LIN {X 0,Y 100.402,Z 358.237,A -85,B 0,C 180,E1 -29156.99,E2 -29156.99} C_VEL
LIN {X 0,Y 100.384,Z 357.85,A -85,B 0,C 180,E1 -29157.993,E2 -29157.993} C_VEL
LIN {X 0,Y 100.386,Z 357.819,A -85,B 0,C 180,E1 -29161.253,E2 -29161.253} C_VEL
LIN {X 0,Y 101.796,Z 362.471,A -85,B 0,C 180,E1 -29171.07,E2 -29171.07} C_VEL
LIN {X 0,Y 103.401,Z 366.135,A -85,B 0,C 180,E1 -29175.775,E2 -29175.775} C_VEL
LIN {X 0,Y 105.074,Z 370.255,A -85,B 0,C 180,E1 -29179.684,E2 -29179.684} C_VEL
LIN {X 0,Y 105.684,Z 372.499,A -85,B 0,C 180,E1 -29181.129,E2 -29181.129} C_VEL
LIN {X 0,Y 106.021,Z 374.366,A -85,B 0,C 180,E1 -29182.034,E2 -29182.034} C_VEL
LIN {X 0,Y 103.387,Z 386.289,A -85,B 0,C 180,E1 -29182.916,E2 -29182.916} C_VEL
LIN {X 0,Y 99.941,Z 396.229,A -85,B 0,C 180,E1 -29183.916,E2 -29183.916} C_VEL
LIN {X 0,Y 96.046,Z 404.883,A -85,B 0,C 180,E1 -29185.113,E2 -29185.113} C_VEL
LIN {X 0,Y 91.456,Z 413.164,A -85,B 0,C 180,E1 -29186.711,E2 -29186.711} C_VEL
LIN {X 0,Y 86.224,Z 421.013,A -85,B 0,C 180,E1 -29188.816,E2 -29188.816} C_VEL
LIN {X 0,Y 80.026,Z 428.854,A -85,B 0,C 180,E1 -29191.798,E2 -29191.798} C_VEL
LIN {X 0,Y 72.277,Z 437.075,A -85,B 0,C 180,E1 -29196.664,E2 -29196.664} C_VEL
LIN {X 0,Y 65.93,Z 442.65,A -85,B 0,C 180,E1 -29201.744,E2 -29201.744} C_VEL
LIN {X 0,Y 59.276,Z 447.852,A -85,B 0,C 180,E1 -29209.305,E2 -29209.305} C_VEL
LIN {X 0,Y 53.929,Z 451.685,A -85,B 0,C 180,E1 -29218.587,E2 -29218.587} C_VEL
LIN {X 0,Y 51.351,Z 453.456,A -85,B 0,C 180,E1 -29225.763,E2 -29225.763} C_VEL
LIN {X 0,Y 49.572,Z 454.73,A -85,B 0,C 180,E1 -29233.533,E2 -29233.533} C_VEL
LIN {X 0,Y 48.724,Z 455.53,A -85,B 0,C 180,E1 -29241.711,E2 -29241.711} C_VEL
LIN {X 0,Y 48.789,Z 455.849,A -85,B 0,C 180,E1 -29250.004,E2 -29250.004} C_VEL
LIN {X 0,Y 48.725,Z 455.516,A -85,B 0,C 180,E1 -29258.297,E2 -29258.297} C_VEL
LIN {X 0,Y 49.574,Z 454.686,A -85,B 0,C 180,E1 -29266.476,E2 -29266.476} C_VEL
LIN {X 0,Y 51.352,Z 453.382,A -85,B 0,C 180,E1 -29274.245,E2 -29274.245} C_VEL
LIN {X 0,Y 55.511,Z 450.407,A -85,B 0,C 180,E1 -29284.736,E2 -29284.736} C_VEL
LIN {X 0,Y 59.279,Z 447.714,A -85,B 0,C 180,E1 -29290.702,E2 -29290.702} C_VEL
LIN {X 0,Y 65.928,Z 442.473,A -85,B 0,C 180,E1 -29298.267,E2 -29298.267} C_VEL
LIN {X 0,Y 73.597,Z 435.578,A -85,B 0,C 180,E1 -29304.266,E2 -29304.266} C_VEL
LIN {X 0,Y 80.378,Z 428.151,A -85,B 0,C 180,E1 -29308.358,E2 -29308.358} C_VEL
LIN {X 0,Y 85.511,Z 421.674,A -85,B 0,C 180,E1 -29310.843,E2 -29310.843} C_VEL
LIN {X 0,Y 90.682,Z 413.947,A -85,B 0,C 180,E1 -29313.038,E2 -29313.038} C_VEL
LIN {X 0,Y 95.26,Z 405.834,A -85,B 0,C 180,E1 -29314.663,E2 -29314.663} C_VEL
LIN {X 0,Y 99.139,Z 397.416,A -85,B 0,C 180,E1 -29315.887,E2 -29315.887} C_VEL
LIN {X 0,Y 102.671,Z 387.658,A -85,B 0,C 180,E1 -29316.868,E2 -29316.868} C_VEL
LIN {X 0,Y 105.515,Z 376.095,A -85,B 0,C 180,E1 -29317.75,E2 -29317.75} C_VEL
LIN {X 0,Y 105.767,Z 374.04,A -85,B 0,C 180,E1 -29317.928,E2 -29317.928} C_VEL
LIN {X 0,Y 105.084,Z 370.805,A -85,B 0,C 180,E1 -29319.661,E2 -29319.661} C_VEL
LIN {X 0,Y 103.427,Z 366.583,A -85,B 0,C 180,E1 -29323.437,E2 -29323.437} C_VEL
LIN {X 0,Y 102.311,Z 364.174,A -85,B 0,C 180,E1 -29326.284,E2 -29326.284} C_VEL
LIN {X 0,Y 101.255,Z 361.634,A -85,B 0,C 180,E1 -29329.818,E2 -29329.818} C_VEL
LIN {X 0,Y 100.146,Z 358.287,A -85,B 0,C 180,E1 -29336.732,E2 -29336.732} C_VEL
LIN {X 0,Y 100.091,Z 357.785,A -85,B 0,C 180,E1 -29337.988,E2 -29337.988} C_VEL
LIN {X 0,Y 100.101,Z 357.82,A -85,B 0,C 180,E1 -29343.019,E2 -29343.019} C_VEL
LIN {X 0,Y 101.129,Z 361.456,A -85,B 0,C 180,E1 -29350.546,E2 -29350.546} C_VEL
LIN {X 0,Y 101.708,Z 362.817,A -85,B 0,C 180,E1 -29352.682,E2 -29352.682} C_VEL
LIN {X 0,Y 103.187,Z 366.252,A -85,B 0,C 180,E1 -29357.049,E2 -29357.049} C_VEL
LIN {X 0,Y 104.694,Z 370.111,A -85,B 0,C 180,E1 -29360.703,E2 -29360.703} C_VEL
LIN {X 0,Y 105.664,Z 373.274,A -85,B 0,C 180,E1 -29363.045,E2 -29363.045} C_VEL
LIN {X 0,Y 103.161,Z 383.593,A -85,B 0,C 180,E1 -29364.046,E2 -29364.046} C_VEL
LIN {X 0,Y 100.108,Z 392.746,A -85,B 0,C 180,E1 -29365.323,E2 -29365.323} C_VEL
LIN {X 0,Y 96.36,Z 401.138,A -85,B 0,C 180,E1 -29366.686,E2 -29366.686} C_VEL
LIN {X 0,Y 92.666,Z 407.987,A -85,B 0,C 180,E1 -29368.152,E2 -29368.152} C_VEL
LIN {X 0,Y 87.652,Z 415.86,A -85,B 0,C 180,E1 -29370.461,E2 -29370.461} C_VEL
LIN {X 0,Y 83.407,Z 421.515,A -85,B 0,C 180,E1 -29372.578,E2 -29372.578} C_VEL
LIN {X 0,Y 77.628,Z 428.233,A -85,B 0,C 180,E1 -29376.073,E2 -29376.073} C_VEL
LIN {X 0,Y 73.727,Z 431.905,A -85,B 0,C 180,E1 -29378.076,E2 -29378.076} C_VEL
LIN {X 0,Y 66.062,Z 437.234,A -85,B 0,C 180,E1 -29380.871,E2 -29380.871} C_VEL
LIN {X 0,Y 58.269,Z 441.79,A -85,B 0,C 180,E1 -29384.678,E2 -29384.678} C_VEL
LIN {X 0,Y 54.358,Z 444.075,A -85,B 0,C 180,E1 -29388.459,E2 -29388.459} C_VEL
LIN {X 0,Y 49.897,Z 446.751,A -85,B 0,C 180,E1 -29395.704,E2 -29395.704} C_VEL
LIN {X 0,Y 46.656,Z 448.491,A -85,B 0,C 180,E1 -29403.129,E2 -29403.129} C_VEL
LIN {X 0,Y 44.155,Z 449.745,A -85,B 0,C 180,E1 -29411.433,E2 -29411.433} C_VEL
LIN {X 0,Y 42.609,Z 450.532,A -85,B 0,C 180,E1 -29420.501,E2 -29420.501} C_VEL
LIN {X 0,Y 42.085,Z 450.831,A -85,B 0,C 180,E1 -29429.995,E2 -29429.995} C_VEL
LIN {X 0,Y 42.608,Z 450.55,A -85,B 0,C 180,E1 -29439.489,E2 -29439.489} C_VEL
LIN {X 0,Y 44.15,Z 449.799,A -85,B 0,C 180,E1 -29448.559,E2 -29448.559} C_VEL
LIN {X 0,Y 46.62,Z 448.583,A -85,B 0,C 180,E1 -29456.883,E2 -29456.883} C_VEL
LIN {X 0,Y 51.76,Z 445.741,A -85,B 0,C 180,E1 -29467.657,E2 -29467.657} C_VEL
LIN {X 0,Y 55.967,Z 443.15,A -85,B 0,C 180,E1 -29473.677,E2 -29473.677} C_VEL
LIN {X 0,Y 63.208,Z 438.053,A -85,B 0,C 180,E1 -29481.102,E2 -29481.102} C_VEL
LIN {X 0,Y 69.847,Z 432.563,A -85,B 0,C 180,E1 -29486.105,E2 -29486.105} C_VEL
LIN {X 0,Y 76.92,Z 425.648,A -85,B 0,C 180,E1 -29490.221,E2 -29490.221} C_VEL
LIN {X 0,Y 83.481,Z 417.714,A -85,B 0,C 180,E1 -29493.436,E2 -29493.436} C_VEL
LIN {X 0,Y 88.75,Z 410.141,A -85,B 0,C 180,E1 -29495.591,E2 -29495.591} C_VEL
LIN {X 0,Y 92.616,Z 403.681,A -85,B 0,C 180,E1 -29496.932,E2 -29496.932} C_VEL
LIN {X 0,Y 96.47,Z 395.828,A -85,B 0,C 180,E1 -29498.251,E2 -29498.251} C_VEL
LIN {X 0,Y 99.737,Z 387.4,A -85,B 0,C 180,E1 -29499.37,E2 -29499.37} C_VEL
LIN {X 0,Y 102.526,Z 377.614,A -85,B 0,C 180,E1 -29500.363,E2 -29500.363} C_VEL
LIN {X 0,Y 102.555,Z 376.884,A -85,B 0,C 180,E1 -29500.653,E2 -29500.653} C_VEL
LIN {X 0,Y 101.635,Z 373.042,A -85,B 0,C 180,E1 -29504.329,E2 -29504.329} C_VEL
LIN {X 0,Y 100.893,Z 370.848,A -85,B 0,C 180,E1 -29507.018,E2 -29507.018} C_VEL
LIN {X 0,Y 100.114,Z 368.403,A -85,B 0,C 180,E1 -29510.657,E2 -29510.657} C_VEL
LIN {X 0,Y 99.502,Z 364.863,A -85,B 0,C 180,E1 -29518.482,E2 -29518.482} C_VEL
LIN {X 0,Y 99.503,Z 365.013,A -85,B 0,C 180,E1 -29521.264,E2 -29521.264} C_VEL
LIN {X 0,Y 100.461,Z 369.199,A -85,B 0,C 180,E1 -29529.945,E2 -29529.945} C_VEL
LIN {X 0,Y 101.631,Z 372.591,A -85,B 0,C 180,E1 -29534.377,E2 -29534.377} C_VEL
LIN {X 0,Y 102.921,Z 376.479,A -85,B 0,C 180,E1 -29538.153,E2 -29538.153} C_VEL
LIN {X 0,Y 103.002,Z 377.05,A -85,B 0,C 180,E1 -29538.524,E2 -29538.524} C_VEL
LIN {X 0,Y 100.454,Z 387.016,A -85,B 0,C 180,E1 -29539.275,E2 -29539.275} C_VEL
LIN {X 0,Y 97.284,Z 395.844,A -85,B 0,C 180,E1 -29540.099,E2 -29540.099} C_VEL
LIN {X 0,Y 93.252,Z 404.495,A -85,B 0,C 180,E1 -29541.155,E2 -29541.155} C_VEL
LIN {X 0,Y 88.492,Z 412.776,A -85,B 0,C 180,E1 -29542.601,E2 -29542.601} C_VEL
LIN {X 0,Y 83.033,Z 420.624,A -85,B 0,C 180,E1 -29544.516,E2 -29544.516} C_VEL
LIN {X 0,Y 77.068,Z 427.848,A -85,B 0,C 180,E1 -29547.032,E2 -29547.032} C_VEL
LIN {X 0,Y 69.679,Z 435.442,A -85,B 0,C 180,E1 -29550.988,E2 -29550.988} C_VEL
LIN {X 0,Y 62.724,Z 441.292,A -85,B 0,C 180,E1 -29555.681,E2 -29555.681} C_VEL
LIN {X 0,Y 56.429,Z 445.925,A -85,B 0,C 180,E1 -29561.65,E2 -29561.65} C_VEL
LIN {X 0,Y 51.851,Z 448.938,A -85,B 0,C 180,E1 -29567.341,E2 -29567.341} C_VEL
LIN {X 0,Y 47.976,Z 451.291,A -85,B 0,C 180,E1 -29574.135,E2 -29574.135} C_VEL
LIN {X 0,Y 44.947,Z 453.063,A -85,B 0,C 180,E1 -29582.031,E2 -29582.031} C_VEL
LIN {X 0,Y 42.797,Z 454.337,A -85,B 0,C 180,E1 -29590.832,E2 -29590.832} C_VEL
LIN {X 0,Y 41.689,Z 455.137,A -85,B 0,C 180,E1 -29600.3,E2 -29600.3} C_VEL
LIN {X 0,Y 41.692,Z 455.457,A -85,B 0,C 180,E1 -29610.005,E2 -29610.005} C_VEL
LIN {X 0,Y 41.69,Z 455.122,A -85,B 0,C 180,E1 -29619.71,E2 -29619.71} C_VEL
LIN {X 0,Y 42.799,Z 454.293,A -85,B 0,C 180,E1 -29629.178,E2 -29629.178} C_VEL
LIN {X 0,Y 44.949,Z 452.988,A -85,B 0,C 180,E1 -29637.979,E2 -29637.979} C_VEL
LIN {X 0,Y 49.822,Z 450.012,A -85,B 0,C 180,E1 -29649.408,E2 -29649.408} C_VEL
LIN {X 0,Y 54.09,Z 447.321,A -85,B 0,C 180,E1 -29655.618,E2 -29655.618} C_VEL
LIN {X 0,Y 61.408,Z 442.077,A -85,B 0,C 180,E1 -29663.244,E2 -29663.244} C_VEL
LIN {X 0,Y 69.684,Z 435.183,A -85,B 0,C 180,E1 -29669.017,E2 -29669.017} C_VEL
LIN {X 0,Y 75.984,Z 428.786,A -85,B 0,C 180,E1 -29672.454,E2 -29672.454} C_VEL
LIN {X 0,Y 82.27,Z 421.277,A -85,B 0,C 180,E1 -29675.189,E2 -29675.189} C_VEL
LIN {X 0,Y 87.699,Z 413.553,A -85,B 0,C 180,E1 -29677.165,E2 -29677.165} C_VEL
LIN {X 0,Y 92.44,Z 405.437,A -85,B 0,C 180,E1 -29678.65,E2 -29678.65} C_VEL
LIN {X 0,Y 96.462,Z 397.019,A -85,B 0,C 180,E1 -29679.731,E2 -29679.731} C_VEL
LIN {X 0,Y 99.499,Z 389.051,A -85,B 0,C 180,E1 -29680.457,E2 -29680.457} C_VEL
LIN {X 0,Y 102.181,Z 379.433,A -85,B 0,C 180,E1 -29681.182,E2 -29681.182} C_VEL
LIN {X 0,Y 102.772,Z 376.736,A -85,B 0,C 180,E1 -29681.433,E2 -29681.433} C_VEL
LIN {X 0,Y 101.62,Z 373.025,A -85,B 0,C 180,E1 -29684.789,E2 -29684.789} C_VEL
LIN {X 0,Y 100.366,Z 369.551,A -85,B 0,C 180,E1 -29689.153,E2 -29689.153} C_VEL
LIN {X 0,Y 99.916,Z 368.232,A -85,B 0,C 180,E1 -29691.277,E2 -29691.277} C_VEL
LIN {X 0,Y 99.189,Z 364.754,A -85,B 0,C 180,E1 -29698.732,E2 -29698.732} C_VEL
LIN {X 0,Y 99.202,Z 364.859,A -85,B 0,C 180,E1 -29702.538,E2 -29702.538} C_VEL
LIN {X 0,Y 99.869,Z 368.268,A -85,B 0,C 180,E1 -29709.696,E2 -29709.696} C_VEL
LIN {X 0,Y 101.258,Z 372.35,A -85,B 0,C 180,E1 -29715.354,E2 -29715.354} C_VEL
LIN {X 0,Y 102.29,Z 376.488,A -85,B 0,C 180,E1 -29719.379,E2 -29719.379} C_VEL
LIN {X 0,Y 102.337,Z 377.035,A -85,B 0,C 180,E1 -29719.71,E2 -29719.71} C_VEL
LIN {X 0,Y 100.312,Z 384.55,A -85,B 0,C 180,E1 -29720.425,E2 -29720.425} C_VEL
LIN {X 0,Y 97.025,Z 393.794,A -85,B 0,C 180,E1 -29721.647,E2 -29721.647} C_VEL
LIN {X 0,Y 93.39,Z 401.547,A -85,B 0,C 180,E1 -29722.807,E2 -29722.807} C_VEL
LIN {X 0,Y 89.544,Z 408.381,A -85,B 0,C 180,E1 -29724.155,E2 -29724.155} C_VEL
LIN {X 0,Y 84.281,Z 416.255,A -85,B 0,C 180,E1 -29726.304,E2 -29726.304} C_VEL
LIN {X 0,Y 79.813,Z 421.909,A -85,B 0,C 180,E1 -29728.286,E2 -29728.286} C_VEL
LIN {X 0,Y 74.088,Z 428.217,A -85,B 0,C 180,E1 -29731.374,E2 -29731.374} C_VEL
LIN {X 0,Y 68.527,Z 433.462,A -85,B 0,C 180,E1 -29734.864,E2 -29734.864} C_VEL
LIN {X 0,Y 63.252,Z 437.837,A -85,B 0,C 180,E1 -29738.938,E2 -29738.938} C_VEL
LIN {X 0,Y 55.986,Z 442.983,A -85,B 0,C 180,E1 -29746.332,E2 -29746.332} C_VEL
LIN {X 0,Y 54.358,Z 444.075,A -85,B 0,C 180,E1 -29748.459,E2 -29748.459} C_VEL
LIN {X 0,Y 50.637,Z 446.185,A -85,B 0,C 180,E1 -29752.92,E2 -29752.92} C_VEL
LIN {X 0,Y 46.435,Z 447.925,A -85,B 0,C 180,E1 -29757.46,E2 -29757.46} C_VEL
LIN {X 0,Y 38.447,Z 450.266,A -85,B 0,C 180,E1 -29769.13,E2 -29769.13} C_VEL
LIN {X 0,Y 35.883,Z 450.882,A -85,B 0,C 180,E1 -29777.367,E2 -29777.367} C_VEL
LIN {X 0,Y 35.442,Z 450.973,A -85,B 0,C 180,E1 -29780.47,E2 -29780.47} C_VEL
LIN {X 0,Y 34.998,Z 451.223,A -85,B 0,C 180,E1 -29789.994,E2 -29789.994} C_VEL
LIN {X 0,Y 35.643,Z 450.94,A -85,B 0,C 180,E1 -29801.366,E2 -29801.366} C_VEL
LIN {X 0,Y 37.52,Z 450.189,A -85,B 0,C 180,E1 -29811.995,E2 -29811.995} C_VEL
LIN {X 0,Y 40.426,Z 448.974,A -85,B 0,C 180,E1 -29821.429,E2 -29821.429} C_VEL
LIN {X 0,Y 46.354,Z 446.131,A -85,B 0,C 180,E1 -29833.015,E2 -29833.015} C_VEL
LIN {X 0,Y 51.071,Z 443.54,A -85,B 0,C 180,E1 -29839.182,E2 -29839.182} C_VEL
LIN {X 0,Y 59.02,Z 438.442,A -85,B 0,C 180,E1 -29846.458,E2 -29846.458} C_VEL
LIN {X 0,Y 66.162,Z 432.952,A -85,B 0,C 180,E1 -29851.198,E2 -29851.198} C_VEL
LIN {X 0,Y 73.66,Z 426.037,A -85,B 0,C 180,E1 -29855.005,E2 -29855.005} C_VEL
LIN {X 0,Y 80.569,Z 418.101,A -85,B 0,C 180,E1 -29857.936,E2 -29857.936} C_VEL
LIN {X 0,Y 86.069,Z 410.528,A -85,B 0,C 180,E1 -29859.882,E2 -29859.882} C_VEL
LIN {X 0,Y 90.049,Z 404.122,A -85,B 0,C 180,E1 -29861.069,E2 -29861.069} C_VEL
LIN {X 0,Y 94.343,Z 395.59,A -85,B 0,C 180,E1 -29862.338,E2 -29862.338} C_VEL
LIN {X 0,Y 97.85,Z 386.64,A -85,B 0,C 180,E1 -29863.37,E2 -29863.37} C_VEL
LIN {X 0,Y 99.213,Z 382.499,A -85,B 0,C 180,E1 -29863.788,E2 -29863.788} C_VEL
LIN {X 0,Y 99.604,Z 380.632,A -85,B 0,C 180,E1 -29864.263,E2 -29864.263} C_VEL
LIN {X 0,Y 98.889,Z 377.185,A -85,B 0,C 180,E1 -29868.446,E2 -29868.446} C_VEL
LIN {X 0,Y 98.533,Z 375.072,A -85,B 0,C 180,E1 -29871.798,E2 -29871.798} C_VEL
LIN {X 0,Y 98.345,Z 371.862,A -85,B 0,C 180,E1 -29878.976,E2 -29878.976} C_VEL
LIN {X 0,Y 98.338,Z 371.997,A -85,B 0,C 180,E1 -29880.639,E2 -29880.639} C_VEL
LIN {X 0,Y 98.892,Z 375.878,A -85,B 0,C 180,E1 -29888.814,E2 -29888.814} C_VEL
LIN {X 0,Y 99.577,Z 378.924,A -85,B 0,C 180,E1 -29893.001,E2 -29893.001} C_VEL
LIN {X 0,Y 99.979,Z 380.711,A -85,B 0,C 180,E1 -29894.939,E2 -29894.939} C_VEL
LIN {X 0,Y 97.288,Z 389.687,A -85,B 0,C 180,E1 -29895.575,E2 -29895.575} C_VEL
LIN {X 0,Y 93.418,Z 399.209,A -85,B 0,C 180,E1 -29896.43,E2 -29896.43} C_VEL
LIN {X 0,Y 87.642,Z 409.922,A -85,B 0,C 180,E1 -29897.786,E2 -29897.786} C_VEL
LIN {X 0,Y 81.96,Z 418.188,A -85,B 0,C 180,E1 -29899.406,E2 -29899.406} C_VEL
LIN {X 0,Y 75.571,Z 425.873,A -85,B 0,C 180,E1 -29901.575,E2 -29901.575} C_VEL
LIN {X 0,Y 69.317,Z 432.203,A -85,B 0,C 180,E1 -29904.154,E2 -29904.154} C_VEL
LIN {X 0,Y 63.294,Z 437.474,A -85,B 0,C 180,E1 -29907.347,E2 -29907.347} C_VEL
LIN {X 0,Y 57.427,Z 441.865,A -85,B 0,C 180,E1 -29911.063,E2 -29911.063} C_VEL
LIN {X 0,Y 49.379,Z 447.07,A -85,B 0,C 180,E1 -29918.489,E2 -29918.489} C_VEL
LIN {X 0,Y 42.397,Z 450.898,A -85,B 0,C 180,E1 -29928.473,E2 -29928.473} C_VEL
LIN {X 0,Y 38.782,Z 452.669,A -85,B 0,C 180,E1 -29937.074,E2 -29937.074} C_VEL
LIN {X 0,Y 36.161,Z 453.945,A -85,B 0,C 180,E1 -29947.133,E2 -29947.133} C_VEL
LIN {X 0,Y 34.707,Z 454.745,A -85,B 0,C 180,E1 -29958.323,E2 -29958.323} C_VEL
LIN {X 0,Y 34.585,Z 455.065,A -85,B 0,C 180,E1 -29970.006,E2 -29970.006} C_VEL
LIN {X 0,Y 34.709,Z 454.73,A -85,B 0,C 180,E1 -29981.688,E2 -29981.688} C_VEL
LIN {X 0,Y 36.163,Z 453.9,A -85,B 0,C 180,E1 -29992.878,E2 -29992.878} C_VEL
LIN {X 0,Y 38.784,Z 452.593,A -85,B 0,C 180,E1 -30002.937,E2 -30002.937} C_VEL
LIN {X 0,Y 44.555,Z 449.619,A -85,B 0,C 180,E1 -30015.227,E2 -30015.227} C_VEL
LIN {X 0,Y 49.383,Z 446.927,A -85,B 0,C 180,E1 -30021.519,E2 -30021.519} C_VEL
LIN {X 0,Y 57.428,Z 441.682,A -85,B 0,C 180,E1 -30028.95,E2 -30028.95} C_VEL
LIN {X 0,Y 66.3,Z 434.788,A -85,B 0,C 180,E1 -30034.299,E2 -30034.299} C_VEL
LIN {X 0,Y 73.739,Z 427.556,A -85,B 0,C 180,E1 -30037.71,E2 -30037.71} C_VEL
LIN {X 0,Y 79.547,Z 420.881,A -85,B 0,C 180,E1 -30039.845,E2 -30039.845} C_VEL
LIN {X 0,Y 85.195,Z 413.157,A -85,B 0,C 180,E1 -30041.569,E2 -30041.569} C_VEL
LIN {X 0,Y 90.102,Z 405.041,A -85,B 0,C 180,E1 -30042.851,E2 -30042.851} C_VEL
LIN {X 0,Y 94.245,Z 396.622,A -85,B 0,C 180,E1 -30043.77,E2 -30043.77} C_VEL
LIN {X 0,Y 97.61,Z 387.893,A -85,B 0,C 180,E1 -30044.461,E2 -30044.461} C_VEL
LIN {X 0,Y 99.726,Z 380.373,A -85,B 0,C 180,E1 -30045.074,E2 -30045.074} C_VEL
LIN {X 0,Y 98.946,Z 377.09,A -85,B 0,C 180,E1 -30048.996,E2 -30048.996} C_VEL
LIN {X 0,Y 98.423,Z 374.847,A -85,B 0,C 180,E1 -30052.564,E2 -30052.564} C_VEL
LIN {X 0,Y 98.038,Z 371.726,A -85,B 0,C 180,E1 -30059.359,E2 -30059.359} C_VEL
LIN {X 0,Y 98.008,Z 371.971,A -85,B 0,C 180,E1 -30062.055,E2 -30062.055} C_VEL
LIN {X 0,Y 98.409,Z 375.692,A -85,B 0,C 180,E1 -30069.841,E2 -30069.841} C_VEL
LIN {X 0,Y 99.023,Z 378.8,A -85,B 0,C 180,E1 -30074.122,E2 -30074.122} C_VEL
LIN {X 0,Y 99.351,Z 380.461,A -85,B 0,C 180,E1 -30075.91,E2 -30075.91} C_VEL
LIN {X 0,Y 98.07,Z 384.948,A -85,B 0,C 180,E1 -30076.555,E2 -30076.555} C_VEL
LIN {X 0,Y 95.174,Z 392.928,A -85,B 0,C 180,E1 -30077.485,E2 -30077.485} C_VEL
LIN {X 0,Y 91.504,Z 400.808,A -85,B 0,C 180,E1 -30078.543,E2 -30078.543} C_VEL
LIN {X 0,Y 86.888,Z 408.776,A -85,B 0,C 180,E1 -30079.892,E2 -30079.892} C_VEL
LIN {X 0,Y 81.394,Z 416.649,A -85,B 0,C 180,E1 -30081.835,E2 -30081.835} C_VEL
LIN {X 0,Y 76.711,Z 422.303,A -85,B 0,C 180,E1 -30083.622,E2 -30083.622} C_VEL
LIN {X 0,Y 70.657,Z 428.611,A -85,B 0,C 180,E1 -30086.46,E2 -30086.46} C_VEL
LIN {X 0,Y 64.743,Z 433.855,A -85,B 0,C 180,E1 -30089.719,E2 -30089.719} C_VEL
LIN {X 0,Y 59.057,Z 438.23,A -85,B 0,C 180,E1 -30093.584,E2 -30093.584} C_VEL
LIN {X 0,Y 51.089,Z 443.376,A -85,B 0,C 180,E1 -30100.829,E2 -30100.829} C_VEL
LIN {X 0,Y 46.37,Z 446.006,A -85,B 0,C 180,E1 -30106.991,E2 -30106.991} C_VEL
LIN {X 0,Y 40.472,Z 448.882,A -85,B 0,C 180,E1 -30118.598,E2 -30118.598} C_VEL
LIN {X 0,Y 37.525,Z 450.136,A -85,B 0,C 180,E1 -30127.996,E2 -30127.996} C_VEL
LIN {X 0,Y 35.442,Z 450.973,A -85,B 0,C 180,E1 -30140.47,E2 -30140.47} C_VEL
LIN {X 0,Y 34.306,Z 451.261,A -85,B 0,C 180,E1 -30150.01,E2 -30150.01} C_VEL
LIN {X 0,Y 32.738,Z 450.99,A -85,B 0,C 180,E1 -30166.819,E2 -30166.819} C_VEL
LIN {X 0,Y 33.895,Z 449.832,A -85,B 0,C 180,E1 -30183.784,E2 -30183.784} C_VEL
LIN {X 0,Y 36.683,Z 448.514,A -85,B 0,C 180,E1 -30192.088,E2 -30192.088} C_VEL
LIN {X 0,Y 44.037,Z 445.376,A -85,B 0,C 180,E1 -30202.927,E2 -30202.927} C_VEL
LIN {X 0,Y 52.467,Z 440.726,A -85,B 0,C 180,E1 -30210.529,E2 -30210.529} C_VEL
LIN {X 0,Y 59.967,Z 435.669,A -85,B 0,C 180,E1 -30215.26,E2 -30215.26} C_VEL
LIN {X 0,Y 66.199,Z 430.719,A -85,B 0,C 180,E1 -30218.261,E2 -30218.261} C_VEL
LIN {X 0,Y 72.547,Z 424.746,A -85,B 0,C 180,E1 -30220.817,E2 -30220.817} C_VEL
LIN {X 0,Y 78.999,Z 417.473,A -85,B 0,C 180,E1 -30223,E2 -30223} C_VEL
LIN {X 0,Y 84.726,Z 409.689,A -85,B 0,C 180,E1 -30224.631,E2 -30224.631} C_VEL
LIN {X 0,Y 88.649,Z 403.371,A -85,B 0,C 180,E1 -30225.551,E2 -30225.551} C_VEL
LIN {X 0,Y 92.898,Z 394.941,A -85,B 0,C 180,E1 -30226.638,E2 -30226.638} C_VEL
LIN {X 0,Y 96.367,Z 386.136,A -85,B 0,C 180,E1 -30227.495,E2 -30227.495} C_VEL
LIN {X 0,Y 96.702,Z 384.376,A -85,B 0,C 180,E1 -30228.471,E2 -30228.471} C_VEL
LIN {X 0,Y 96.608,Z 382.315,A -85,B 0,C 180,E1 -30231.634,E2 -30231.634} C_VEL
LIN {X 0,Y 96.667,Z 379.04,A -85,B 0,C 180,E1 -30238.958,E2 -30238.958} C_VEL
LIN {X 0,Y 96.696,Z 378.99,A -85,B 0,C 180,E1 -30240.26,E2 -30240.26} C_VEL
LIN {X 0,Y 96.851,Z 382.493,A -85,B 0,C 180,E1 -30247.819,E2 -30247.819} C_VEL
LIN {X 0,Y 97.126,Z 384.2,A -85,B 0,C 180,E1 -30250.424,E2 -30250.424} C_VEL
LIN {X 0,Y 96.746,Z 386.119,A -85,B 0,C 180,E1 -30251.302,E2 -30251.302} C_VEL
LIN {X 0,Y 93.36,Z 395.071,A -85,B 0,C 180,E1 -30251.882,E2 -30251.882} C_VEL
LIN {X 0,Y 89.116,Z 403.721,A -85,B 0,C 180,E1 -30252.607,E2 -30252.607} C_VEL
LIN {X 0,Y 84.059,Z 411.999,A -85,B 0,C 180,E1 -30253.617,E2 -30253.617} C_VEL
LIN {X 0,Y 78.211,Z 419.846,A -85,B 0,C 180,E1 -30254.997,E2 -30254.997} C_VEL
LIN {X 0,Y 70.88,Z 427.963,A -85,B 0,C 180,E1 -30257.143,E2 -30257.143} C_VEL
LIN {X 0,Y 61.943,Z 435.902,A -85,B 0,C 180,E1 -30260.614,E2 -30260.614} C_VEL
LIN {X 0,Y 54.1,Z 441.474,A -85,B 0,C 180,E1 -30264.593,E2 -30264.593} C_VEL
LIN {X 0,Y 45.286,Z 446.677,A -85,B 0,C 180,E1 -30271.41,E2 -30271.41} C_VEL
LIN {X 0,Y 37.357,Z 450.505,A -85,B 0,C 180,E1 -30281.199,E2 -30281.199} C_VEL
LIN {X 0,Y 33.021,Z 452.276,A -85,B 0,C 180,E1 -30290.328,E2 -30290.328} C_VEL
LIN {X 0,Y 29.719,Z 453.552,A -85,B 0,C 180,E1 -30301.781,E2 -30301.781} C_VEL
LIN {X 0,Y 27.779,Z 454.353,A -85,B 0,C 180,E1 -30315.353,E2 -30315.353} C_VEL
LIN {X 0,Y 27.477,Z 454.672,A -85,B 0,C 180,E1 -30330.008,E2 -30330.008} C_VEL
LIN {X 0,Y 27.78,Z 454.337,A -85,B 0,C 180,E1 -30344.662,E2 -30344.662} C_VEL
LIN {X 0,Y 29.722,Z 453.506,A -85,B 0,C 180,E1 -30358.232,E2 -30358.232} C_VEL
LIN {X 0,Y 33.024,Z 452.198,A -85,B 0,C 180,E1 -30369.684,E2 -30369.684} C_VEL
LIN {X 0,Y 39.869,Z 449.225,A -85,B 0,C 180,E1 -30382.498,E2 -30382.498} C_VEL
LIN {X 0,Y 45.291,Z 446.532,A -85,B 0,C 180,E1 -30388.598,E2 -30388.598} C_VEL
LIN {X 0,Y 54.102,Z 441.288,A -85,B 0,C 180,E1 -30395.42,E2 -30395.42} C_VEL
LIN {X 0,Y 63.529,Z 434.391,A -85,B 0,C 180,E1 -30400.115,E2 -30400.115} C_VEL
LIN {X 0,Y 71.624,Z 426.873,A -85,B 0,C 180,E1 -30403.082,E2 -30403.082} C_VEL
LIN {X 0,Y 78.215,Z 419.46,A -85,B 0,C 180,E1 -30405.013,E2 -30405.013} C_VEL
LIN {X 0,Y 84.055,Z 411.526,A -85,B 0,C 180,E1 -30406.417,E2 -30406.417} C_VEL
LIN {X 0,Y 89.831,Z 401.866,A -85,B 0,C 180,E1 -30407.553,E2 -30407.553} C_VEL
LIN {X 0,Y 95.071,Z 390.031,A -85,B 0,C 180,E1 -30408.379,E2 -30408.379} C_VEL
LIN {X 0,Y 96.761,Z 385.188,A -85,B 0,C 180,E1 -30408.678,E2 -30408.678} C_VEL
LIN {X 0,Y 96.896,Z 384.114,A -85,B 0,C 180,E1 -30409.342,E2 -30409.342} C_VEL
LIN {X 0,Y 96.44,Z 381.405,A -85,B 0,C 180,E1 -30413.725,E2 -30413.725} C_VEL
LIN {X 0,Y 96.446,Z 378.596,A -85,B 0,C 180,E1 -30420,E2 -30420} C_VEL
LIN {X 0,Y 96.354,Z 378.932,A -85,B 0,C 180,E1 -30421.568,E2 -30421.568} C_VEL
LIN {X 0,Y 96.342,Z 382.031,A -85,B 0,C 180,E1 -30428.39,E2 -30428.39} C_VEL
LIN {X 0,Y 96.468,Z 384.495,A -85,B 0,C 180,E1 -30432.091,E2 -30432.091} C_VEL
LIN {X 0,Y 96.081,Z 385.975,A -85,B 0,C 180,E1 -30432.576,E2 -30432.576} C_VEL
LIN {X 0,Y 92.649,Z 394.792,A -85,B 0,C 180,E1 -30433.51,E2 -30433.51} C_VEL
LIN {X 0,Y 88.568,Z 402.871,A -85,B 0,C 180,E1 -30434.426,E2 -30434.426} C_VEL
LIN {X 0,Y 83.928,Z 410.394,A -85,B 0,C 180,E1 -30435.627,E2 -30435.627} C_VEL
LIN {X 0,Y 78.219,Z 418.059,A -85,B 0,C 180,E1 -30437.312,E2 -30437.312} C_VEL
LIN {X 0,Y 71,Z 426.071,A -85,B 0,C 180,E1 -30439.879,E2 -30439.879} C_VEL
LIN {X 0,Y 63.098,Z 433.082,A -85,B 0,C 180,E1 -30443.226,E2 -30443.226} C_VEL
LIN {X 0,Y 55.455,Z 438.623,A -85,B 0,C 180,E1 -30447.477,E2 -30447.477} C_VEL
LIN {X 0,Y 46.765,Z 443.768,A -85,B 0,C 180,E1 -30454.245,E2 -30454.245} C_VEL
LIN {X 0,Y 41.465,Z 446.398,A -85,B 0,C 180,E1 -30460.288,E2 -30460.288} C_VEL
LIN {X 0,Y 34.622,Z 449.274,A -85,B 0,C 180,E1 -30472.477,E2 -30472.477} C_VEL
LIN {X 0,Y 31.069,Z 450.527,A -85,B 0,C 180,E1 -30483.094,E2 -30483.094} C_VEL
LIN {X 0,Y 28.477,Z 451.365,A -85,B 0,C 180,E1 -30498.183,E2 -30498.183} C_VEL
LIN {X 0,Y 27.918,Z 451.614,A -85,B 0,C 180,E1 -30509.993,E2 -30509.993} C_VEL
LIN {X 0,Y 28.737,Z 451.331,A -85,B 0,C 180,E1 -30524.149,E2 -30524.149} C_VEL
LIN {X 0,Y 31.063,Z 450.579,A -85,B 0,C 180,E1 -30536.896,E2 -30536.896} C_VEL
LIN {X 0,Y 36.683,Z 448.514,A -85,B 0,C 180,E1 -30552.088,E2 -30552.088} C_VEL
LIN {X 0,Y 40.003,Z 447.04,A -85,B 0,C 180,E1 -30559.055,E2 -30559.055} C_VEL
LIN {X 0,Y 45.159,Z 444.006,A -85,B 0,C 180,E1 -30569.763,E2 -30569.763} C_VEL
LIN {X 0,Y 51.219,Z 440.151,A -85,B 0,C 180,E1 -30577.928,E2 -30577.928} C_VEL
LIN {X 0,Y 55.611,Z 437.316,A -85,B 0,C 180,E1 -30580.89,E2 -30580.89} C_VEL
LIN {X 0,Y 63.916,Z 431.108,A -85,B 0,C 180,E1 -30584.166,E2 -30584.166} C_VEL
LIN {X 0,Y 70.534,Z 425.135,A -85,B 0,C 180,E1 -30586.273,E2 -30586.273} C_VEL
LIN {X 0,Y 77.228,Z 417.86,A -85,B 0,C 180,E1 -30588.024,E2 -30588.024} C_VEL
LIN {X 0,Y 83.133,Z 410.076,A -85,B 0,C 180,E1 -30589.334,E2 -30589.334} C_VEL
LIN {X 0,Y 87.513,Z 403.125,A -85,B 0,C 180,E1 -30590.123,E2 -30590.123} C_VEL
LIN {X 0,Y 91.743,Z 394.835,A -85,B 0,C 180,E1 -30591.003,E2 -30591.003} C_VEL
LIN {X 0,Y 93.634,Z 390.6,A -85,B 0,C 180,E1 -30591.366,E2 -30591.366} C_VEL
LIN {X 0,Y 94.071,Z 388.852,A -85,B 0,C 180,E1 -30592.487,E2 -30592.487} C_VEL
LIN {X 0,Y 94.564,Z 385.937,A -85,B 0,C 180,E1 -30600,E2 -30600} C_VEL
LIN {X 0,Y 94.35,Z 389.054,A -85,B 0,C 180,E1 -30606.953,E2 -30606.953} C_VEL
LIN {X 0,Y 94.181,Z 389.734,A -85,B 0,C 180,E1 -30607.291,E2 -30607.291} C_VEL
LIN {X 0,Y 89.045,Z 401.242,A -85,B 0,C 180,E1 -30607.944,E2 -30607.944} C_VEL
LIN {X 0,Y 83.539,Z 410.379,A -85,B 0,C 180,E1 -30608.711,E2 -30608.711} C_VEL
LIN {X 0,Y 77.538,Z 418.434,A -85,B 0,C 180,E1 -30609.717,E2 -30609.717} C_VEL
LIN {X 0,Y 71.572,Z 425.093,A -85,B 0,C 180,E1 -30610.919,E2 -30610.919} C_VEL
LIN {X 0,Y 64.81,Z 431.423,A -85,B 0,C 180,E1 -30612.605,E2 -30612.605} C_VEL
LIN {X 0,Y 58.148,Z 436.692,A -85,B 0,C 180,E1 -30614.795,E2 -30614.795} C_VEL
LIN {X 0,Y 51.548,Z 441.083,A -85,B 0,C 180,E1 -30617.389,E2 -30617.389} C_VEL
LIN {X 0,Y 42.017,Z 446.285,A -85,B 0,C 180,E1 -30623.092,E2 -30623.092} C_VEL
LIN {X 0,Y 33.099,Z 450.112,A -85,B 0,C 180,E1 -30631.872,E2 -30631.872} C_VEL
LIN {X 0,Y 27.909,Z 451.883,A -85,B 0,C 180,E1 -30640.946,E2 -30640.946} C_VEL
LIN {X 0,Y 23.684,Z 453.159,A -85,B 0,C 180,E1 -30653.607,E2 -30653.607} C_VEL
LIN {X 0,Y 20.967,Z 453.96,A -85,B 0,C 180,E1 -30670.426,E2 -30670.426} C_VEL
LIN {X 0,Y 20.364,Z 454.279,A -85,B 0,C 180,E1 -30690.01,E2 -30690.01} C_VEL
LIN {X 0,Y 20.969,Z 453.944,A -85,B 0,C 180,E1 -30709.593,E2 -30709.593} C_VEL
LIN {X 0,Y 23.688,Z 453.112,A -85,B 0,C 180,E1 -30726.408,E2 -30726.408} C_VEL
LIN {X 0,Y 27.913,Z 451.804,A -85,B 0,C 180,E1 -30739.067,E2 -30739.067} C_VEL
LIN {X 0,Y 35.975,Z 448.831,A -85,B 0,C 180,E1 -30751.548,E2 -30751.548} C_VEL
LIN {X 0,Y 42.022,Z 446.138,A -85,B 0,C 180,E1 -30756.916,E2 -30756.916} C_VEL
LIN {X 0,Y 51.552,Z 440.894,A -85,B 0,C 180,E1 -30762.624,E2 -30762.624} C_VEL
LIN {X 0,Y 61.127,Z 434.277,A -85,B 0,C 180,E1 -30766.27,E2 -30766.27} C_VEL
LIN {X 0,Y 69.888,Z 426.479,A -85,B 0,C 180,E1 -30768.662,E2 -30768.662} C_VEL
LIN {X 0,Y 76.687,Z 419.065,A -85,B 0,C 180,E1 -30770.138,E2 -30770.138} C_VEL
LIN {X 0,Y 82.678,Z 411.131,A -85,B 0,C 180,E1 -30771.193,E2 -30771.193} C_VEL
LIN {X 0,Y 88.855,Z 400.977,A -85,B 0,C 180,E1 -30772.061,E2 -30772.061} C_VEL
LIN {X 0,Y 93.572,Z 390.55,A -85,B 0,C 180,E1 -30772.583,E2 -30772.583} C_VEL
LIN {X 0,Y 93.938,Z 389.52,A -85,B 0,C 180,E1 -30772.635,E2 -30772.635} C_VEL
LIN {X 0,Y 94.118,Z 388.771,A -85,B 0,C 180,E1 -30773.029,E2 -30773.029} C_VEL
LIN {X 0,Y 94.334,Z 385.615,A -85,B 0,C 180,E1 -30780,E2 -30780} C_VEL
LIN {X 0,Y 93.861,Z 387.962,A -85,B 0,C 180,E1 -30786.449,E2 -30786.449} C_VEL
LIN {X 0,Y 93.776,Z 389.279,A -85,B 0,C 180,E1 -30788.621,E2 -30788.621} C_VEL
LIN {X 0,Y 88.569,Z 400.657,A -85,B 0,C 180,E1 -30789.688,E2 -30789.688} C_VEL
LIN {X 0,Y 83.993,Z 408.34,A -85,B 0,C 180,E1 -30790.514,E2 -30790.514} C_VEL
LIN {X 0,Y 78.096,Z 416.42,A -85,B 0,C 180,E1 -30791.847,E2 -30791.847} C_VEL
LIN {X 0,Y 72.214,Z 423.09,A -85,B 0,C 180,E1 -30793.28,E2 -30793.28} C_VEL
LIN {X 0,Y 65.58,Z 429.398,A -85,B 0,C 180,E1 -30795.302,E2 -30795.302} C_VEL
LIN {X 0,Y 59.023,Z 434.64,A -85,B 0,C 180,E1 -30797.706,E2 -30797.706} C_VEL
LIN {X 0,Y 52.567,Z 439.015,A -85,B 0,C 180,E1 -30800.619,E2 -30800.619} C_VEL
LIN {X 0,Y 43.179,Z 444.16,A -85,B 0,C 180,E1 -30806.455,E2 -30806.455} C_VEL
LIN {X 0,Y 37.273,Z 446.791,A -85,B 0,C 180,E1 -30811.942,E2 -30811.942} C_VEL
LIN {X 0,Y 29.333,Z 449.665,A -85,B 0,C 180,E1 -30824.035,E2 -30824.035} C_VEL
LIN {X 0,Y 24.975,Z 450.918,A -85,B 0,C 180,E1 -30835.74,E2 -30835.74} C_VEL
LIN {X 0,Y 21.933,Z 451.705,A -85,B 0,C 180,E1 -30851.301,E2 -30851.301} C_VEL
LIN {X 0,Y 20.838,Z 452.004,A -85,B 0,C 180,E1 -30869.99,E2 -30869.99} C_VEL
LIN {X 0,Y 21.931,Z 451.722,A -85,B 0,C 180,E1 -30888.681,E2 -30888.681} C_VEL
LIN {X 0,Y 24.969,Z 450.969,A -85,B 0,C 180,E1 -30904.249,E2 -30904.249} C_VEL
LIN {X 0,Y 31.566,Z 448.975,A -85,B 0,C 180,E1 -30920.325,E2 -30920.325} C_VEL
LIN {X 0,Y 40.166,Z 445.766,A -85,B 0,C 180,E1 -30931.018,E2 -30931.018} C_VEL
LIN {X 0,Y 49.365,Z 441.117,A -85,B 0,C 180,E1 -30937.717,E2 -30937.717} C_VEL
LIN {X 0,Y 55.611,Z 437.316,A -85,B 0,C 180,E1 -30940.89,E2 -30940.89} C_VEL
LIN {X 0,Y 59.961,Z 434.198,A -85,B 0,C 180,E1 -30943.422,E2 -30943.422} C_VEL
LIN {X 0,Y 66.27,Z 428.681,A -85,B 0,C 180,E1 -30948.326,E2 -30948.326} C_VEL
LIN {X 0,Y 72.385,Z 422.453,A -85,B 0,C 180,E1 -30952.181,E2 -30952.181} C_VEL
LIN {X 0,Y 74.909,Z 419.637,A -85,B 0,C 180,E1 -30953.032,E2 -30953.032} C_VEL
LIN {X 0,Y 76.181,Z 418.124,A -85,B 0,C 180,E1 -30953.25,E2 -30953.25} C_VEL
LIN {X 0,Y 82.119,Z 410.462,A -85,B 0,C 180,E1 -30954.186,E2 -30954.186} C_VEL
LIN {X 0,Y 86.615,Z 403.45,A -85,B 0,C 180,E1 -30954.75,E2 -30954.75} C_VEL
LIN {X 0,Y 90.964,Z 395.093,A -85,B 0,C 180,E1 -30955.43,E2 -30955.43} C_VEL
LIN {X 0,Y 91.328,Z 394.289,A -85,B 0,C 180,E1 -30955.586,E2 -30955.586} C_VEL
LIN {X 0,Y 91.947,Z 392.775,A -85,B 0,C 180,E1 -30960,E2 -30960} C_VEL
LIN {X 0,Y 91.498,Z 394.299,A -85,B 0,C 180,E1 -30963.149,E2 -30963.149} C_VEL
LIN {X 0,Y 86.816,Z 403.482,A -85,B 0,C 180,E1 -30963.49,E2 -30963.49} C_VEL
LIN {X 0,Y 81.889,Z 411.224,A -85,B 0,C 180,E1 -30963.933,E2 -30963.933} C_VEL
LIN {X 0,Y 75.788,Z 419.068,A -85,B 0,C 180,E1 -30964.567,E2 -30964.567} C_VEL
LIN {X 0,Y 68.837,Z 426.416,A -85,B 0,C 180,E1 -30965.511,E2 -30965.511} C_VEL
LIN {X 0,Y 60.91,Z 433.283,A -85,B 0,C 180,E1 -30966.842,E2 -30966.842} C_VEL
LIN {X 0,Y 51.601,Z 439.73,A -85,B 0,C 180,E1 -30969.121,E2 -30969.121} C_VEL
LIN {X 0,Y 43.116,Z 444.357,A -85,B 0,C 180,E1 -30972.059,E2 -30972.059} C_VEL
LIN {X 0,Y 36.448,Z 447.372,A -85,B 0,C 180,E1 -30975.418,E2 -30975.418} C_VEL
LIN {X 0,Y 29.952,Z 449.719,A -85,B 0,C 180,E1 -30980.21,E2 -30980.21} C_VEL
LIN {X 0,Y 23.857,Z 451.491,A -85,B 0,C 180,E1 -30987.92,E2 -30987.92} C_VEL
LIN {X 0,Y 18.449,Z 452.767,A -85,B 0,C 180,E1 -31000.386,E2 -31000.386} C_VEL
LIN {X 0,Y 14.468,Z 453.567,A -85,B 0,C 180,E1 -31020.955,E2 -31020.955} C_VEL
LIN {X 0,Y 13.272,Z 453.888,A -85,B 0,C 180,E1 -31050.016,E2 -31050.016} C_VEL
LIN {X 0,Y 14.472,Z 453.551,A -85,B 0,C 180,E1 -31079.07,E2 -31079.07} C_VEL
LIN {X 0,Y 18.454,Z 452.719,A -85,B 0,C 180,E1 -31099.631,E2 -31099.631} C_VEL
LIN {X 0,Y 23.863,Z 451.411,A -85,B 0,C 180,E1 -31112.093,E2 -31112.093} C_VEL
LIN {X 0,Y 33.178,Z 448.436,A -85,B 0,C 180,E1 -31122.428,E2 -31122.428} C_VEL
LIN {X 0,Y 39.774,Z 445.744,A -85,B 0,C 180,E1 -31126.393,E2 -31126.393} C_VEL
LIN {X 0,Y 49.894,Z 440.5,A -85,B 0,C 180,E1 -31130.431,E2 -31130.431} C_VEL
LIN {X 0,Y 58.849,Z 434.617,A -85,B 0,C 180,E1 -31132.695,E2 -31132.695} C_VEL
LIN {X 0,Y 67.112,Z 427.79,A -85,B 0,C 180,E1 -31134.206,E2 -31134.206} C_VEL
LIN {X 0,Y 74.925,Z 419.695,A -85,B 0,C 180,E1 -31135.327,E2 -31135.327} C_VEL
LIN {X 0,Y 81.021,Z 411.968,A -85,B 0,C 180,E1 -31136.02,E2 -31136.02} C_VEL
LIN {X 0,Y 85.596,Z 404.988,A -85,B 0,C 180,E1 -31136.444,E2 -31136.444} C_VEL
LIN {X 0,Y 89.74,Z 397.339,A -85,B 0,C 180,E1 -31136.731,E2 -31136.731} C_VEL
LIN {X 0,Y 90.62,Z 395.45,A -85,B 0,C 180,E1 -31136.802,E2 -31136.802} C_VEL
LIN {X 0,Y 91.445,Z 393.485,A -85,B 0,C 180,E1 -31137.635,E2 -31137.635} C_VEL
LIN {X 0,Y 91.735,Z 392.49,A -85,B 0,C 180,E1 -31140,E2 -31140} C_VEL
LIN {X 0,Y 91.138,Z 393.945,A -85,B 0,C 180,E1 -31144.423,E2 -31144.423} C_VEL
LIN {X 0,Y 90.204,Z 395.998,A -85,B 0,C 180,E1 -31144.777,E2 -31144.777} C_VEL
LIN {X 0,Y 85.602,Z 404.591,A -85,B 0,C 180,E1 -31145.346,E2 -31145.346} C_VEL
LIN {X 0,Y 79.544,Z 413.63,A -85,B 0,C 180,E1 -31146.269,E2 -31146.269} C_VEL
LIN {X 0,Y 72.653,Z 421.783,A -85,B 0,C 180,E1 -31147.444,E2 -31147.444} C_VEL
LIN {X 0,Y 65.801,Z 428.378,A -85,B 0,C 180,E1 -31148.883,E2 -31148.883} C_VEL
LIN {X 0,Y 57.271,Z 435.032,A -85,B 0,C 180,E1 -31150.954,E2 -31150.954} C_VEL
LIN {X 0,Y 50.512,Z 439.407,A -85,B 0,C 180,E1 -31153.092,E2 -31153.092} C_VEL
LIN {X 0,Y 40.526,Z 444.552,A -85,B 0,C 180,E1 -31157.465,E2 -31157.465} C_VEL
LIN {X 0,Y 34.06,Z 447.183,A -85,B 0,C 180,E1 -31161.778,E2 -31161.778} C_VEL
LIN {X 0,Y 24.932,Z 450.057,A -85,B 0,C 180,E1 -31172.242,E2 -31172.242} C_VEL
LIN {X 0,Y 19.54,Z 451.309,A -85,B 0,C 180,E1 -31183.985,E2 -31183.985} C_VEL
LIN {X 0,Y 15.409,Z 452.096,A -85,B 0,C 180,E1 -31202.849,E2 -31202.849} C_VEL
LIN {X 0,Y 13.75,Z 452.396,A -85,B 0,C 180,E1 -31229.985,E2 -31229.985} C_VEL
LIN {X 0,Y 15.406,Z 452.112,A -85,B 0,C 180,E1 -31257.127,E2 -31257.127} C_VEL
LIN {X 0,Y 19.533,Z 451.359,A -85,B 0,C 180,E1 -31276.006,E2 -31276.006} C_VEL
LIN {X 0,Y 24.906,Z 450.144,A -85,B 0,C 180,E1 -31287.823,E2 -31287.823} C_VEL
LIN {X 0,Y 34.047,Z 447.303,A -85,B 0,C 180,E1 -31298.245,E2 -31298.245} C_VEL
LIN {X 0,Y 40.514,Z 444.709,A -85,B 0,C 180,E1 -31302.554,E2 -31302.554} C_VEL
LIN {X 0,Y 50.492,Z 439.609,A -85,B 0,C 180,E1 -31306.972,E2 -31306.972} C_VEL
LIN {X 0,Y 58.952,Z 434.117,A -85,B 0,C 180,E1 -31309.568,E2 -31309.568} C_VEL
LIN {X 0,Y 67.491,Z 427.201,A -85,B 0,C 180,E1 -31311.574,E2 -31311.574} C_VEL
LIN {X 0,Y 75.214,Z 419.263,A -85,B 0,C 180,E1 -31313.096,E2 -31313.096} C_VEL
LIN {X 0,Y 76.181,Z 418.124,A -85,B 0,C 180,E1 -31313.25,E2 -31313.25} C_VEL
LIN {X 0,Y 75.815,Z 418.486,A -85,B 0,C 180,E1 -31314.001,E2 -31314.001} C_VEL
LIN {X 0,Y 74.849,Z 419.543,A -85,B 0,C 180,E1 -31314.69,E2 -31314.69} C_VEL
LIN {X 0,Y 69.41,Z 425.082,A -85,B 0,C 180,E1 -31316.844,E2 -31316.844} C_VEL
LIN {X 0,Y 62.202,Z 431.441,A -85,B 0,C 180,E1 -31319.034,E2 -31319.034} C_VEL
LIN {X 0,Y 57.85,Z 434.798,A -85,B 0,C 180,E1 -31320.159,E2 -31320.159} C_VEL
LIN {X 0,Y 53.302,Z 437.876,A -85,B 0,C 180,E1 -31320.949,E2 -31320.949} C_VEL
LIN {X 0,Y 42.205,Z 443.964,A -85,B 0,C 180,E1 -31322.533,E2 -31322.533} C_VEL
LIN {X 0,Y 35.23,Z 446.979,A -85,B 0,C 180,E1 -31324.177,E2 -31324.177} C_VEL
LIN {X 0,Y 28.292,Z 449.327,A -85,B 0,C 180,E1 -31326.533,E2 -31326.533} C_VEL
LIN {X 0,Y 21.463,Z 451.098,A -85,B 0,C 180,E1 -31330.842,E2 -31330.842} C_VEL
LIN {X 0,Y 14.856,Z 452.373,A -85,B 0,C 180,E1 -31338.929,E2 -31338.929} C_VEL
LIN {X 0,Y 8.938,Z 453.174,A -85,B 0,C 180,E1 -31358.197,E2 -31358.197} C_VEL
LIN {X 0,Y 6.164,Z 453.495,A -85,B 0,C 180,E1 -31410.034,E2 -31410.034} C_VEL
LIN {X 0,Y 8.944,Z 453.158,A -85,B 0,C 180,E1 -31461.833,E2 -31461.833} C_VEL
LIN {X 0,Y 14.862,Z 452.325,A -85,B 0,C 180,E1 -31481.084,E2 -31481.084} C_VEL
LIN {X 0,Y 21.47,Z 451.016,A -85,B 0,C 180,E1 -31489.166,E2 -31489.166} C_VEL
LIN {X 0,Y 31.762,Z 448.042,A -85,B 0,C 180,E1 -31494.766,E2 -31494.766} C_VEL
LIN {X 0,Y 38.722,Z 445.349,A -85,B 0,C 180,E1 -31496.688,E2 -31496.688} C_VEL
LIN {X 0,Y 49.214,Z 440.107,A -85,B 0,C 180,E1 -31498.605,E2 -31498.605} C_VEL
LIN {X 0,Y 59.483,Z 433.406,A -85,B 0,C 180,E1 -31499.78,E2 -31499.78} C_VEL
LIN {X 0,Y 68.528,Z 425.687,A -85,B 0,C 180,E1 -31500.398,E2 -31500.398} C_VEL
LIN {X 0,Y 75.562,Z 418.273,A -85,B 0,C 180,E1 -31500.829,E2 -31500.829} C_VEL
LIN {X 0,Y 77.321,Z 416.223,A -85,B 0,C 180,E1 -31500.923,E2 -31500.923} C_VEL
LIN {X 0,Y 77.332,Z 416.193,A -85,B 0,C 180,E1 -31501.322,E2 -31501.322} C_VEL
LIN {X 0,Y 70.326,Z 423.876,A -85,B 0,C 180,E1 -31501.998,E2 -31501.998} C_VEL
LIN {X 0,Y 63.333,Z 430.185,A -85,B 0,C 180,E1 -31502.833,E2 -31502.833} C_VEL
LIN {X 0,Y 56.357,Z 435.424,A -85,B 0,C 180,E1 -31503.883,E2 -31503.883} C_VEL
LIN {X 0,Y 49.392,Z 439.799,A -85,B 0,C 180,E1 -31505.063,E2 -31505.063} C_VEL
LIN {X 0,Y 38.992,Z 444.943,A -85,B 0,C 180,E1 -31507.508,E2 -31507.508} C_VEL
LIN {X 0,Y 32.115,Z 447.574,A -85,B 0,C 180,E1 -31509.974,E2 -31509.974} C_VEL
LIN {X 0,Y 21.988,Z 450.448,A -85,B 0,C 180,E1 -31516.455,E2 -31516.455} C_VEL
LIN {X 0,Y 15.481,Z 451.7,A -85,B 0,C 180,E1 -31524.749,E2 -31524.749} C_VEL
LIN {X 0,Y 9.662,Z 452.487,A -85,B 0,C 180,E1 -31543.298,E2 -31543.298} C_VEL
LIN {X 0,Y 6.685,Z 452.786,A -85,B 0,C 180,E1 -31589.969,E2 -31589.969} C_VEL
LIN {X 0,Y 9.656,Z 452.503,A -85,B 0,C 180,E1 -31636.673,E2 -31636.673} C_VEL
LIN {X 0,Y 15.474,Z 451.75,A -85,B 0,C 180,E1 -31655.25,E2 -31655.25} C_VEL
LIN {X 0,Y 21.965,Z 450.535,A -85,B 0,C 180,E1 -31663.686,E2 -31663.686} C_VEL
LIN {X 0,Y 32.105,Z 447.693,A -85,B 0,C 180,E1 -31670.053,E2 -31670.053} C_VEL
LIN {X 0,Y 38.98,Z 445.099,A -85,B 0,C 180,E1 -31672.539,E2 -31672.539} C_VEL
LIN {X 0,Y 49.379,Z 440,A -85,B 0,C 180,E1 -31675.017,E2 -31675.017} C_VEL
LIN {X 0,Y 58.088,Z 434.507,A -85,B 0,C 180,E1 -31676.464,E2 -31676.464} C_VEL
LIN {X 0,Y 66.821,Z 427.59,A -85,B 0,C 180,E1 -31677.59,E2 -31677.59} C_VEL
LIN {X 0,Y 74.695,Z 419.65,A -85,B 0,C 180,E1 -31678.486,E2 -31678.486} C_VEL
LIN {X 0,Y 77.324,Z 416.601,A -85,B 0,C 180,E1 -31678.709,E2 -31678.709} C_VEL
LIN {X 0,Y 77.313,Z 416.632,A -85,B 0,C 180,E1 -31679.123,E2 -31679.123} C_VEL
LIN {X 0,Y 70.279,Z 424.314,A -85,B 0,C 180,E1 -31679.476,E2 -31679.476} C_VEL
LIN {X 0,Y 63.248,Z 430.642,A -85,B 0,C 180,E1 -31679.926,E2 -31679.926} C_VEL
LIN {X 0,Y 56.223,Z 435.908,A -85,B 0,C 180,E1 -31680.6,E2 -31680.6} C_VEL
LIN {X 0,Y 53.302,Z 437.876,A -85,B 0,C 180,E1 -31680.949,E2 -31680.949} C_VEL
LIN {X 0,Y 52.42,Z 439.538,A -85,B 0,C 180,E1 -31681.05,E2 -31681.05} C_VEL
LIN {X 0,Y 52.42,Z 600,A -85,B 0,C 180,E1 -31681.05,E2 -31681.05} C_VEL
LIN {X 0,Y 52.42,Z 600,A -85,B 0,C 180,E1 -31681.05,E2 -31681.05}

QRS_NEXT_CUT()

QRS_NEXT()
QRS_HOME()

END
